TYPE EcCoeSdo_Par_Write_typ : 	
	STRUCT  (*parameter structure*)
		
        nSubIndex       : BYTE; 
        nIndex          : WORD;
        pSrcBuf         : POINTER TO DWORD; 
        cbBufLen        : UDINT; 
        tTimeout        : TIME := DEFAULT_ADS_TIMEOUT ;

	END_STRUCT
END_TYPE

(* stored: Version 1.1.0.1, ProductVersion 3.1.4024.3
   DUT EcCoeSdo_Par_Write_typ: Id {955b64c1-4559-0d66-1b1a-674c8634539d} *)
